{attribute 'GeneratedUsingTerminal: EK1100-0000-0018'}
{attribute addProperty BoxType "EK1100-0000-0018"}
{attribute addProperty Id "Beckhoff_ER8xxxEK1122Beckhoff_ER8xxxEK1122_33861AE064"}
{attribute addProperty CRC "393564351"}
{attribute addProperty Size "64"}
TYPE Beckhoff_ER8xxx_177550BF EXTENDS EK1100_1FC0878B :
STRUCT
	{attribute addProperty Name "Beckhoff_ER8xxxEK1122"}
	{attribute addProperty PreviousPort "Beckhoff ER8xxx : B"}
	Beckhoff_ER8xxxEK1122 : Beckhoff_ER8xxxEK1122_33861AE0;
END_STRUCT
END_TYPE

(* stored: Version 1.2.0.0, ProductVersion 3.1.4024.9
   DUT Beckhoff_ER8xxx_177550BF: Id {375df43c-e924-4f24-bc64-1e1e5175c99a} *)
